
DATA_BLOCK DB304
    STRUCT
        LEITURA: ARRAY[0 .. 0] OF WORD;
    END_STRUCT
BEGIN
END_DATA_BLOCK
